// Brief: Setup Arm Adjust
FUNCTION_BLOCK PUBLIC FB_SetupCtrlManualAdjust EXTENDS FB_SetupArmCtrlBase
VAR
	// friction compensation scale
	m_frictionScale :LREAL :=0.5;
	
	// velocity threshold for friction compensation 
	m_jnt3FrictionCompVelLow :LREAL := 0.0005;
	m_frictionScaleLow :LREAL :=0.1;
	m_jnt3FrictionCompVelMiddle :LREAL := 0.005;
	m_frictionScaleMiddle :LREAL :=0.2;
	m_jnt3FrictionCompVelHigh :LREAL := 0.05;
	m_frictionScaleHigh :LREAL :=0.3;

	// distance buffer from joint limit to start damp
	m_limitBufferForDamp :LREAL :=0.05;
	
	// max damp
	m_maxDamp : LREAL := 1000;
	
	// joint velocity threshold for coulomb friction transition
	m_cFrictionVelThres : LREAL := 5.0 * g_deg2Rad;
	
	m_limitBufferForCtrl : LREAL := 0.00;
END_VAR

// override this function in each exact controller
METHOD PROTECTED calcCmdJntPos : BOOL
VAR_IN_OUT CONSTANT
	i_setupArm	:FB_SetupArm;
END_VAR


VAR 
	i :INT;
	caliJntIdx :INT;
END_VAR
FOR i:= 1 TO 4 DO
	m_jntEnableFlag[i] := BOOL_TO_INT( NOT (SafetyCheck.m_SafetyCheck.m_jntErrFlag[i_setupArm.armIdx, 0, 3] OR  SafetyCheck.m_SafetyCheck.m_jntErrFlag[i_setupArm.armIdx, i, 3]));
	IF m_jntOPMode[i] = DriverOPMode_Trq THEN
		m_cmdJntPos[i]:=i_setupArm.curJntPos[i];
	END_IF
END_FOR
END_METHOD

// override this function in each exact controller
METHOD PROTECTED calcCmdJntTrq : BOOL
VAR_IN_OUT CONSTANT
	i_setupArm	:FB_SetupArm;
END_VAR
VAR
	i:INT;
	vel :LREAL;
	scale:LREAL;
	ratio:LREAL;
	dampScale :LREAL;
	limitDis:LREAL;
	dampOffset : LREAL;
	transitScale:LREAL;
	cFriction:LREAL;
END_VAR
// set joint torque to zero in default
m_cmdJntTrq := g_zeroVec5d;

// friction scale
vel:=ABS(i_setupArm.curJntVel[3]);
IF vel < m_jnt3FrictionCompVelLow THEN
	m_frictionScale := m_frictionScaleLow * vel/m_jnt3FrictionCompVelLow ;
ELSIF  vel > m_jnt3FrictionCompVelLow AND vel  < m_jnt3FrictionCompVelMiddle THEN
	ratio:= (vel-m_jnt3FrictionCompVelLow)/(m_jnt3FrictionCompVelMiddle-m_jnt3FrictionCompVelLow);
	m_frictionScale :=m_frictionScaleLow+ratio * (m_frictionScaleMiddle-m_frictionScaleLow);
ELSIF  vel > m_jnt3FrictionCompVelMiddle AND vel  < m_jnt3FrictionCompVelHigh THEN
	ratio:= (vel-m_jnt3FrictionCompVelMiddle)/(m_jnt3FrictionCompVelHigh-m_jnt3FrictionCompVelMiddle);
	m_frictionScale :=m_frictionScaleMiddle+ratio * (m_frictionScaleHigh-m_frictionScaleMiddle);
ELSIF  vel > m_jnt3FrictionCompVelHigh THEN
	m_frictionScale := m_frictionScaleHigh;
END_IF

// add damp near joint limit 
//IF (i_setupArm.curJntPos[3] > GVL_SetupMotorParameters.g_maxJntPos[1,3] - m_limitBufferForCtrl ) 
//	OR (i_setupArm.curJntPos[3] < GVL_SetupMotorParameters.g_minJntPos[1,3] + m_limitBufferForCtrl) THEN// OR CartControl.m_cartRobot.m_slaveCart.m_columnAdjustEnable
	//dampOffset:= 0;
IF (i_setupArm.curJntPos[3] > GVL_SetupMotorParameters.g_maxJntPos[1,3] - m_limitBufferForDamp AND  i_setupArm.curJntVel[3]> 0 ) 
	OR (i_setupArm.curJntPos[3] < GVL_SetupMotorParameters.g_minJntPos[1,3] + m_limitBufferForDamp AND  i_setupArm.curJntVel[3]<0 )  THEN
	limitDis := MIN(GVL_SetupMotorParameters.g_maxJntPos[1,3] - i_setupArm.curJntPos[3], i_setupArm.curJntPos[3]-GVL_SetupMotorParameters.g_minJntPos[1,3]);
	dampScale  :=LIMIT(0, 1-limitDis/(m_limitBufferForDamp-m_limitBufferForCtrl),1);
	dampOffset:=-dampScale * m_maxDamp * i_setupArm.curJntVel[3];
END_IF

// add friction compensation for joint3
m_frictionScale := LIMIT(0, m_frictionScale, 1);
m_cmdJntTrq[3]:=LIMIT(-g_largeNum, m_frictionScale * sign(i_setupArm.curJntVel[3])*jnt3Friction(i_setupArm.armIdx, i_setupArm.curJntPos[3])+ dampOffset,30);

//add friction compensation for joint4
transitScale := LIMIT(0, ABS(i_setupArm.curJntVel[4]/m_cFrictionVelThres),1);
cFriction:= transitScale * sign(i_setupArm.curJntVel[4]) * GVL_SetupArmDynamics.g_setupJnt4Friction[i_setupArm.armIdx];
m_cmdJntTrq[4]:= m_cmdJntTrq[4]+cFriction;
END_METHOD

METHOD PUBLIC init : BOOL
VAR_IN_OUT CONSTANT
	i_setupArm	:FB_SetupArm;
END_VAR
VAR_IN_OUT 
	r_setupArmCtrlCmd :ST_SetupArmCtrlCmds;
END_VAR
VAR
	i:INT;
END_VAR
SUPER^.Init(i_setupArm,r_setupArmCtrlCmd);

// disable joints if this joint is an unrecoverable failure
FOR i:=1 TO 4 DO
	m_jntEnableFlag[i] := BOOL_TO_INT( NOT (SafetyCheck.m_SafetyCheck.m_jntErrFlag[i_setupArm.armIdx, 0, 3] OR  SafetyCheck.m_SafetyCheck.m_jntErrFlag[i_setupArm.armIdx, i, 3]));
	m_jntOPMode[i]:=DriverOPMode_Trq;
	m_cmdJntPos[i] := i_setupArm.curJntPos[i];
END_FOR
END_METHOD

METHOD PROTECTED jnt3Friction : Lreal
VAR_INPUT
	i_armIdx:INT;
	i_jnt3Pos :LREAL;
END_VAR

VAR
	q:LREAL;
END_VAR
q := LIMIT(GVL_SetupArmDynamics.g_setupJnt3GravityPosRange[i_armIdx,1], i_jnt3Pos, GVL_SetupArmDynamics.g_setupJnt3GravityPosRange[i_armIdx,2]);
jnt3Friction:=GVL_SetupArmDynamics.g_setupJnt3FrictionParams[i_armIdx,1]*EXPT(q,3)+GVL_SetupArmDynamics.g_setupJnt3FrictionParams[i_armIdx,2]*EXPT(q,2)+
				GVL_SetupArmDynamics.g_setupJnt3FrictionParams[i_armIdx,3]*q+GVL_SetupArmDynamics.g_setupJnt3FrictionParams[i_armIdx,4];
END_METHOD

END_FUNCTION_BLOCK

(* stored: Version 1.1.0.1, ProductVersion 3.1.4024.11
   POU FB_SetupCtrlManualAdjust: Id {a66618bf-53b6-41ea-9ead-5a7cf0054c7f}, SpecialFunc None
   Method calcCmdJntPos: Id {a3473076-af2e-4c76-847c-85354c287698}
   Method calcCmdJntTrq: Id {c618bd90-4444-4b54-b7cd-0646bf55f729}
   Method init: Id {f9e2fdef-c3dd-4598-8bef-00a8d9aa9850}
   Method jnt3Friction: Id {e5cc270a-8755-465e-9228-86a9a255b090} *)
